// Mitsubishi GX Works2 project: 0308   PLC: Q03UDE

PROGRAM ai
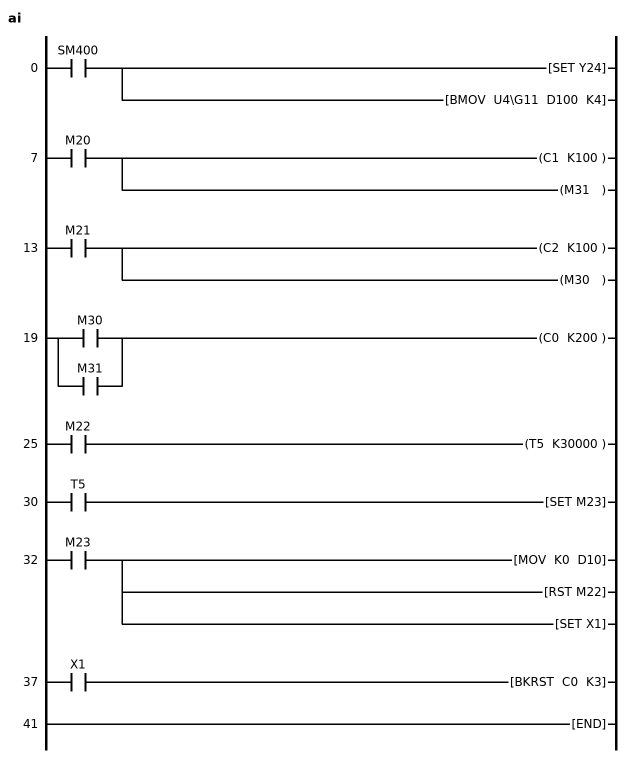
0     LD      SM400
      SET     Y24
      BMOV    U4\G11 D100 K4
7     LD      M20
      OUT     C1 K100
      OUT     M31
13    LD      M21
      OUT     C2 K100
      OUT     M30
19    LD      M30
      OR      M31
      OUT     C0 K200
25    LD      M22
      OUT     T5 K30000
30    LD      T5
      SET     M23
32    LD      M23
      MOV     K0 D10
      RST     M22
      SET     X1
37    LD      X1
      BKRST   C0 K3
41    END
END_PROGRAM

PROGRAM invert
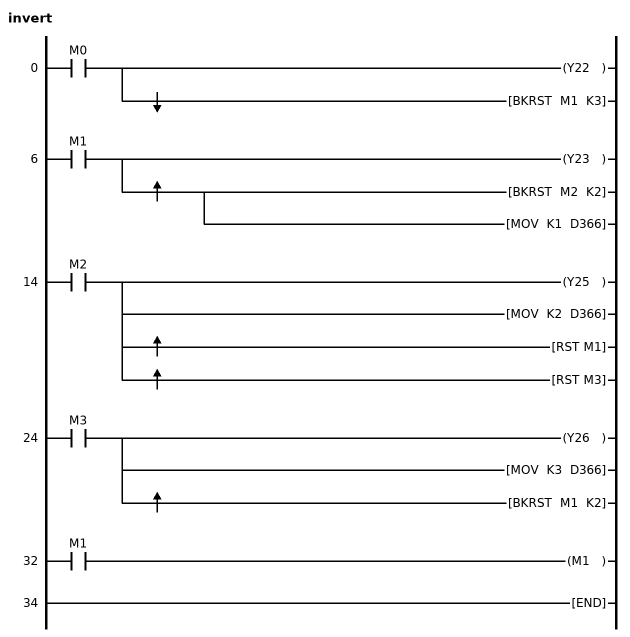
0     LD      M0
      OUT     Y22
      MEF
      BKRST   M1 K3
6     LD      M1
      OUT     Y23
      MEP
      BKRST   M2 K2
      MOV     K1 D366
14    LD      M2
      OUT     Y25
      MOV     K2 D366
      MPS
      MEP
      RST     M1
      MPP
      MEP
      RST     M3
24    LD      M3
      OUT     Y26
      MOV     K3 D366
      MEP
      BKRST   M1 K2
32    LD      M1
      OUT     M1
34    END
END_PROGRAM

PROGRAM LIGHT
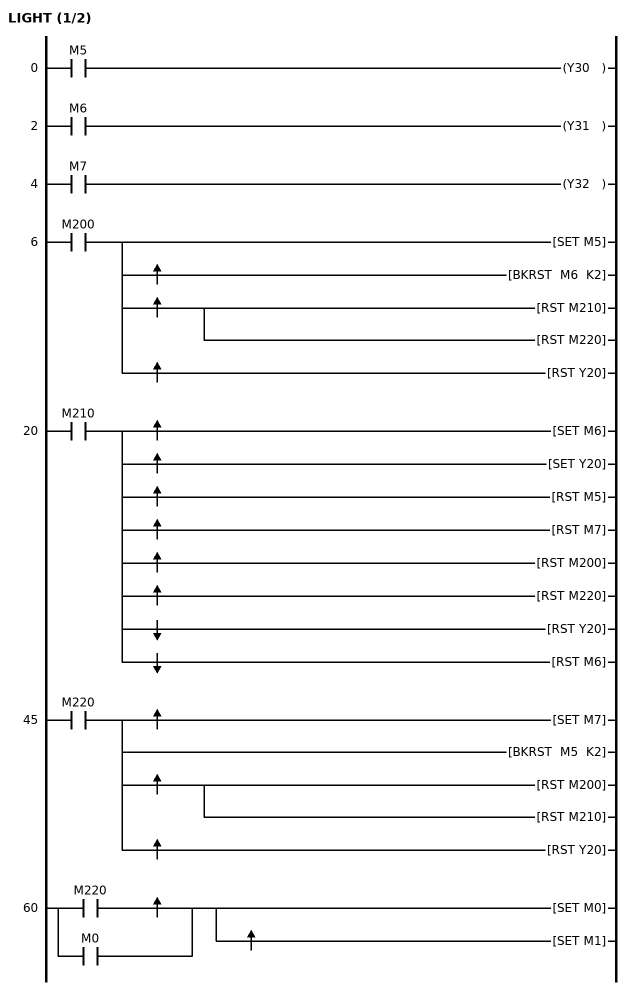
0     LD      M5
      OUT     Y30
2     LD      M6
      OUT     Y31
4     LD      M7
      OUT     Y32
6     LD      M200
      SET     M5
      MPS
      MEP
      BKRST   M6 K2
      MRD
      MEP
      RST     M210
      RST     M220
      MPP
      MEP
      RST     Y20
20    LD      M210
      MPS
      MEP
      SET     M6
      MRD
      MEP
      SET     Y20
      MRD
      MEP
      RST     M5
      MRD
      MEP
      RST     M7
      MRD
      MEP
      RST     M200
      MRD
      MEP
      RST     M220
      MRD
      MEF
      RST     Y20
      MPP
      MEF
      RST     M6
45    LD      M220
      MPS
      MEP
      SET     M7
      MPP
      BKRST   M5 K2
      MPS
      MEP
      RST     M200
      RST     M210
      MPP
      MEP
      RST     Y20
60    LD      M220
      MEP
      OR      M0
      SET     M0
      MEP
      SET     M1
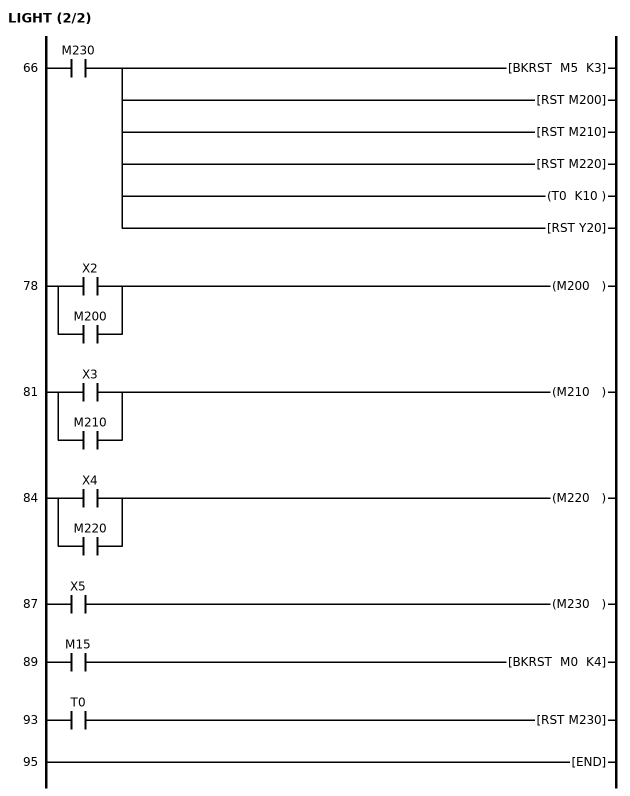
66    LD      M230
      BKRST   M5 K3
      RST     M200
      RST     M210
      RST     M220
      OUT     T0 K10
      RST     Y20
78    LD      X2
      OR      M200
      OUT     M200
81    LD      X3
      OR      M210
      OUT     M210
84    LD      X4
      OR      M220
      OUT     M220
87    LD      X5
      OUT     M230
89    LD      M15
      BKRST   M0 K4
93    LD      T0
      RST     M230
95    END
END_PROGRAM
